INTERFACE I_PreCheckedNode EXTENDS I_Node

METHOD PreExecutionCheck
VAR_INPUT
	Check : I_PreExecutionChecks;
END_VAR
END_METHOD

END_INTERFACE

(* stored: Version 1.1.0.1, ProductVersion 3.1.4024.15
   Itf I_PreCheckedNode: Id {47dfb7b8-9827-0c5a-0039-24de36ca0aae}
   Method PreExecutionCheck: Id {f6c9e145-e3fb-0e01-24ef-03a2e185fc1d} *)
